FUNCTION "CLEAR_LS_1" : Void
{ S7_Optimized_Access := 'TRUE' }
VERSION : 0.1
   VAR_IN_OUT
      IN : "t_LString";
   END_VAR


BEGIN
	#IN.Len := 0;
END_FUNCTION

